Staubli VAL3: OnF4.pgx

program OnF4()
begin
  //
  PublicData:bSimulaiton=true
  call Motion:AllMotion(sItem)
  bUserRefresh=true
end
